INTERFACE I_ErrorSource EXTENDS I_HasAdsError, I_HasGenericError, I_HasError

END_INTERFACE

(* stored: Version 1.1.0.1, ProductVersion 3.1.4024.14
   Itf I_ErrorSource: Id {bca4a0af-4bb7-0b31-008f-9e4c6b49bc9a} *)
